FUNCTION_BLOCK Train_Gate
  (* Standard: 61499-2 *)
  (* Version 0.1, 2015-00-14, Th?o, PC_THEO *)
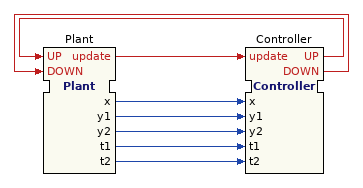
  FBS
    Plant : Plant;
    Controller : Controller;
  END_FBS
  EVENT_CONNECTIONS
    Plant.update TO Controller.update;
    Controller.UP TO Plant.UP;
    Controller.DOWN TO Plant.DOWN;
  END_CONNECTIONS
  DATA_CONNECTIONS
    Plant.x TO Controller.x;
    Plant.y1 TO Controller.y1;
    Plant.y2 TO Controller.y2;
    Plant.t1 TO Controller.t1;
    Plant.t2 TO Controller.t2;
  END_CONNECTIONS
END_FUNCTION_BLOCK
